Fanuc KAREL source: kb00015.compact.KL

PROGRAM KB00015
%STACKSIZE=65535
%PRIORITY=65535
%NOLOCKGROUP
VAR
P1 : STRING[80]
P2 : INTEGER
BEGIN
P1='A'
P2=1
CALL_PROG(P1,P2)
END KB00015
